{attribute 'linkalways'} 
{attribute 'no_explicit_call' := 'This FB is a CLASS and must be accessed using methods or properties'}
{attribute 'enable_dynamic_creation'}
FUNCTION_BLOCK _TcVnVector2_INT EXTENDS AliasDatatypeBase
VAR
	localData : TcVnVector2_INT;
	activeData : REFERENCE TO TcVnVector2_INT REF= localData;
	aliasBaseDatatype : _Array0to1OfINT;
END_VAR

PROPERTY PUBLIC Address : PVOID
GET
Address := ADR(activeData);
END_GET
END_PROPERTY

METHOD PUBLIC ClearReference
VAR_INPUT
END_VAR
activeData REF= localData;
SetBaseDatatypeReference();
END_METHOD

METHOD PUBLIC Clone : I_Datatype
VAR
    pClone : POINTER TO _TcVnVector2_INT;
END_VAR
pClone := __NEW(_TcVnVector2_INT);
Clone := pClone^;
END_METHOD

METHOD FB_init : BOOL
VAR_INPUT
	bInitRetains : BOOL; // if TRUE, the retain variables are initialized (warm start / cold start)
	bInCopyCode : BOOL;  // if TRUE, the instance afterwards gets moved into the copy code (online change)
	//InitialValue : <type>; // if possible, not all values can be initialized
END_VAR
//localData := InitialValue; // if possible, not all values can be initialized
SetBaseDatatypeReference();
AddBaseDatatype(aliasBaseDatatype);
END_METHOD

PROPERTY PUBLIC Identifier : T_MAXSTRING
GET
Identifier := 'TcVnVector2_INT';
END_GET
END_PROPERTY

METHOD PUBLIC MakeReferenceTo
VAR_INPUT
	ReferenceTarget : REFERENCE TO TcVnVector2_INT;
END_VAR
activeData REF= ReferenceTarget;
SetBaseDatatypeReference();
END_METHOD

METHOD PROTECTED SetBaseDatatypeReference
VAR_INPUT
END_VAR
aliasBaseDatatype.MakeReferenceTo(activeData);
END_METHOD

PROPERTY PUBLIC Size : UDINT
GET
Size := SIZEOF(activeData);
END_GET
END_PROPERTY

METHOD TryMakeReferenceTo : BOOL
VAR_INPUT
	Target : I_Datatype;
END_VAR
VAR
	targetAsAlias : I_AliasDatatype;
	pTargetData : POINTER TO TcVnVector2_INT;
END_VAR
IF NOT Target.TryResolveAsAliasDatatype(targetAsAlias) THEN
	RETURN;
END_IF

IF targetAsAlias.Identifier <> Identifier THEN
	RETURN;
END_IF

pTargetData := Target.Address;
activeData REF= pTargetData^;
SetBaseDatatypeReference();
TryMakeReferenceTo := TRUE;
END_METHOD

PROPERTY PUBLIC Value : REFERENCE TO TcVnVector2_INT
GET
Value REF= activeData;
END_GET
END_PROPERTY

END_FUNCTION_BLOCK

(* stored: Version 1.1.0.1, ProductVersion 3.1.4024.13
   POU _TcVnVector2_INT: Id {4d0e7e07-b601-08cc-0b29-a3ec117f90c2}, SpecialFunc None
   Folder Core: Id {8aa41d9b-7567-0f34-1b70-4f32dd1a6710}
   Folder Protected: Id {f75df117-0c26-073b-0860-a72d75d4b0ef}
   Folder Customize: Id {de1c652e-35dd-055f-2cc9-24165f422da9}
   Folder Constructor: Id {4350d3ca-e26c-045e-1135-6becca0607bf}
   Property Address: Id {38745c24-311e-0bc4-38c5-d05481eb98c2}
   Get Get: Id {7782900b-4dd0-026d-3bcb-1daa84eec5a2}
   Method ClearReference: Id {323ecaae-bfd5-0001-0122-a0942446f391}
   Method Clone: Id {994000c8-7972-083a-30a1-547236e89055}
   Method FB_init: Id {108d0fea-447b-0fda-2c59-309f7c48be70}
   Property Identifier: Id {97e996dd-2648-0df6-0803-a6f7a79ce90c}
   Get Get: Id {d4b5d91c-5785-09dc-10bf-fefb987664b0}
   Method MakeReferenceTo: Id {3679879f-02e1-0f54-20d4-d15dceb43e2f}
   Method SetBaseDatatypeReference: Id {ac700500-6766-09a3-2072-149cf0264d05}
   Property Size: Id {85375cc8-36ff-0998-0217-29843c9b527c}
   Get Get: Id {566780b2-898c-0c63-27c6-4b1074caa573}
   Method TryMakeReferenceTo: Id {22038eef-0ffe-0eef-2c8d-da27263d71b2}
   Property Value: Id {41813faf-00e3-0c6b-3c7d-faf3573fdf3a}
   Get Get: Id {31d5759e-996e-0dcb-345c-70c3fcd191a0} *)
